FUNCTION_BLOCK SpeedSpFlowSensorFail (* Basic Function Block Type *)
  (* Standard: 61499-2 *)
  (* Version 0.0, 7/20/2026, Schneider Electric, Template *)
  PACKAGE SE.Nereda;
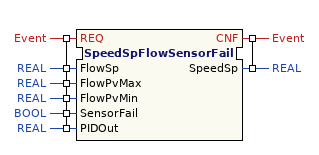
  EVENT_INPUT
    REQ WITH FlowPvMax, FlowPvMin, SensorFail, FlowSp, PIDOut;
  END_EVENT
  EVENT_OUTPUT
    CNF WITH SpeedSp;
  END_EVENT
  VAR_INPUT
    FlowSp : REAL;
    FlowPvMax : REAL;
    FlowPvMin : REAL;
    SensorFail : BOOL;
    PIDOut : REAL;
  END_VAR
  VAR_OUTPUT
    SpeedSp : REAL;
  END_VAR
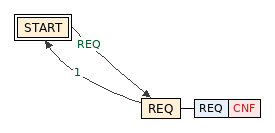
  EC_STATES
    START; (* Initial State *)
    REQ : REQ -> CNF; (* Normal execution *)
  END_STATES
  EC_TRANSITIONS
    START TO REQ := REQ;
    REQ TO START := 1;
  END_TRANSITIONS
  ALGORITHM REQ IN ST: (* Normally executed algorithm *)
;
IF NOT SensorFail THEN
	SpeedSp := PIDOut;
ELSE
	SpeedSp := (FlowSp - FlowPvMin)/(FlowPvMax - FlowPvMin) * 100;
END_IF;
  END_ALGORITHM
END_FUNCTION_BLOCK
